TYPE "UDT_All_Data_symap"
VERSION : 0.1
  STRUCT
    Wincc : "UDT_Wincc";   // Вложенный чистый UDT для WinCC (In, Out)
    In :  "UDT_Symap_In";          // Данные чтения
    Raw : "UDT_Symap_Analog_Reals"; // Мгновенные значения входов  отмасштабируемые

  END_STRUCT;
END_TYPE
